//NOTE：this block would stop checking once a trigger is detected. 
//	re-init this block if want to start another check
FUNCTION_BLOCK FB_MSCtrlTriggerCheck
VAR_INPUT
END_VAR
VAR_OUTPUT
END_VAR
VAR
	// flag if master-slave control is enabled
	m_MSCtrlTrigger :BOOL;
	
	// block run time
	m_timePeriod :LREAL;
	
	// gripper state: 0-init, 1-open, 2-close, 3-reopen, 1-2-3 for one grip action
	m_gripperState :INT;
	
	// grip action counts
	m_gripActionCounts :INT;

	// two grip action within this duration indication to enable master-slave control
	m_checkDuration : LREAL;
	
	// time cycle
	m_timeCycle :LREAL;
	
	// time stamp for first grip
	m_firstGripTime :LREAL;
	
	// angle threshold indicating gripper open
	m_openAngThres :LREAL := g_maxGripAngle * 0.7;
	
	// angle threshold indicating gripper close
	m_closeAngThres :LREAL := 5.0 *g_deg2rad;
END_VAR

METHOD gripActionCheck : BOOL
VAR_INPUT
	i_gripAngle :LREAL;
END_VAR
gripActionCheck:=false;
CASE m_gripperState OF 
	0:
		IF i_gripAngle > m_openAngThres THEN
			m_gripperState :=1;
		END_IF
		
	1: IF i_gripAngle < m_openAngThres AND i_gripAngle > m_closeAngThres THEN
			m_gripperState:=2;
		END_IF
		
	2:
		IF i_gripAngle < m_closeAngThres THEN
			m_gripperState :=3;
		ELSIF i_gripAngle > m_openAngThres THEN
			m_gripperState :=1;
		END_IF
	3:
		IF i_gripAngle > m_openAngThres THEN
			m_gripperState :=4;
		END_IF
	4:
		gripActionCheck:=TRUE;
		m_gripperState:=0;
END_CASE
END_METHOD

METHOD init : BOOL
VAR_INPUT
	i_timeCycle :LREAL;
	i_checkDuration :LREAL;
END_VAR
m_timeCycle :=i_timeCycle;
m_checkDuration := i_checkDuration;
m_gripperState:=0;
m_gripActionCounts:=0;
m_MSCtrlTrigger :=false;
END_METHOD

METHOD reset : BOOL
VAR_INPUT
END_VAR
m_gripperState:=0;
m_gripActionCounts:=0;
m_MSCtrlTrigger :=FALSE;
END_METHOD

METHOD run : BOOL
VAR_INPUT
	i_gripAngle :LREAL;
END_VAR
IF m_MSCtrlTrigger THEN
	run := TRUE;
	RETURN;
END_IF

m_timePeriod := m_timePeriod + m_timeCycle;

// detect one grip action
IF gripActionCheck(i_gripAngle) THEN
	m_gripActionCounts:=m_gripActionCounts+1;
	
	// first grip
	IF 1=m_gripActionCounts THEN
		m_firstGripTime := m_timePeriod;
	ELSIF m_gripActionCounts>=2 THEN
		// second grip and trigger success
		IF m_timePeriod - m_firstGripTime < m_checkDuration THEN
			m_MSCtrlTrigger :=TRUE;
		ELSE
		// set second grip as new first one
			m_gripActionCounts:=1;
			m_firstGripTime:=m_timePeriod;
		END_IF
	END_IF
END_IF


run :=FALSE;
END_METHOD

END_FUNCTION_BLOCK

(* stored: Version 1.1.0.1, ProductVersion 3.1.4024.12
   POU FB_MSCtrlTriggerCheck: Id {636c1ff6-aa47-444d-ac82-ac1207a0e0c5}, SpecialFunc None
   Method gripActionCheck: Id {f4d967c1-2379-40e6-9da8-88bd04c5294b}
   Method init: Id {018ed218-08b5-486a-a90f-59216f36b894}
   Method reset: Id {daea767c-bf3c-41b3-8be1-c82ba8609916}
   Method run: Id {81d1deb4-e804-44ce-bcbb-550e871aa806} *)
